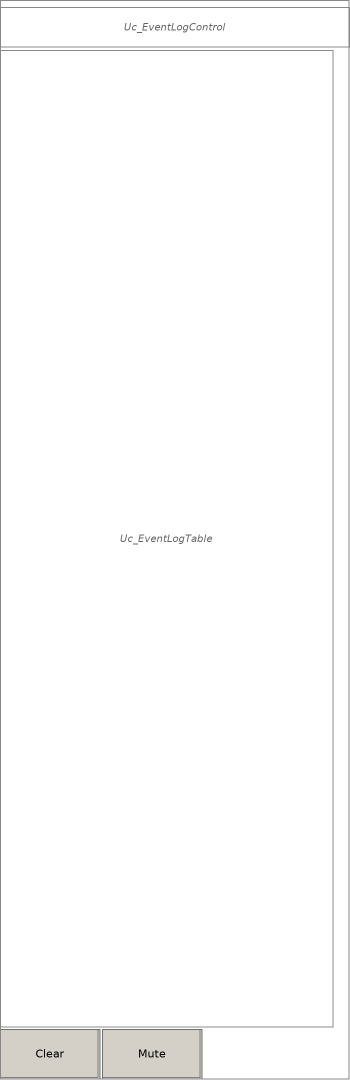
VISUALIZATION Uc_EventLog  // 350x1080
    Frame (0,50 333x977)
        shows Uc_EventLogTable(stVisu := stTable)
    Button (0,1029 100x50), "Clear"
        tap stControl.bQuittAll
    Button (102,1029 100x50), "Mute"
        tap stControl.bMute
    Frame (0,7 350x40)
        shows Uc_EventLogControl(stVisu := stControl)
END_VISUALIZATION

(* stored: Version 1.1.0.1
   Visu Uc_EventLog: Id {b9993396-44eb-41ac-83c8-33ce283c282c} *)
